SUBAPPLICATION AR2_TAP_TO_AR (* Zapft einen zusaetzlichen Nur-Lese-Pfad (AR_OUT, plain AR) aus einer bestehenden AR2-Verbindung ab, ohne deren urspruengliche Persistenz-/Restore-Kette zu unterbrechen. Socket AR2_IN haengt an die Quelle (einen bestehenden AR2-Plug, z.B. AR_CALIBRATE_2P_REF.X_LOW), Plug AR2_OUT fuehrt die AR2-Verbindung unveraendert zum urspruenglichen Ziel weiter (einen bestehenden AR2-Socket, z.B. INI_AR2.VAL). Kombination aus AR2_TO_AR + AR_SPLIT_2 + AR_TO_AR2 (3 bereits vorhandene Standardbausteine) - kein eigener AR2-Split-Baustein existiert im Projekt, AR2 ist wie jeder Adapter strikt 1:1. *)
  (* Standard: 61499-2; Description: Copyright (c) 2026 Meisterschulen am Ostbahnhof This program and the accompanying materials are made available under the terms of the Eclipse Public License 2.0 which is available at https://www.eclipse.org/legal/epl-2.0/ SPDX-License-Identifier: EPL-2.0 *)
  (* Version 1.0, 2026-09-20, Franz Höpfinger, Meisterschulen am Ostbahnhof, initial implementation - fuer die Rohwert-Anzeige (Zero/Span bzw. Min/Mid/Max Raw) in logiBUS_AI_Calibrate_IDA_OPC/_3P_IDA_OPC (Button_AI_Calibrate_OPC_UA/_3P_OPC_UA): AR_CALIBRATE_2P_REF/_3P_REF speichern X_LOW/X_HIGH bzw. X_MIN/X_MID/X_MAX bereits als AR2-Plugs, bisher aber nur an die INI-Persistierung angeschlossen, nirgends zur Anzeige. *)
  PACKAGE MyLib::sys;
  (* Documentation:
  AR2_TAP_TO_AR
   🇩🇪 Deutsch
   Haengt zwischen eine bestehende AR2-Plug/Socket-Verbindung, ohne deren Verhalten zu aendern, und liefert zusaetzlich einen Nur-Lese-Spiegel (AR_OUT, plain AR) des aktuellen Werts.
   Warum nicht einfach splitten?
   Adapter sind strikt 1:1 - ein Plug wie AR_CALIBRATE_2P_REF.X_LOW kann nur an EINEN Socket angeschlossen werden. Fuer unidirektionale Adapter (AR/AX) gibt es dafuer AR_SPLIT_2/AX_SPLIT_2 usw. - fuer bidirektionale AR2 existiert kein aequivalenter Split-Baustein im Projekt, da AR2 normalerweise genau 1 Erzeuger und genau 1 Verbraucher hat.
   Wie es funktioniert
   AR2_TO_AR (Socket AR2_BIDIR, haengt an die Quelle) spiegelt die von der Quelle geschriebene Seite nach AR_OUT - dieser Wert wird per AR_SPLIT_2 aufgeteilt: einmal nach aussen (AR_OUT dieses Bausteins, fuer die Anzeige), einmal in AR_TO_AR2 (Socket AR_IN), das daraus wieder eine vollwertige AR2-Verbindung macht (Plug AR2_BIDIR, geht weiter zum urspruenglichen Ziel, z.B. INI_AR2). Der Rueckweg (persistierter/restaurierter Wert von INI_AR2) laeuft symmetrisch zurueck: AR_TO_AR2.AR_OUT speist AR2_TO_AR.AR_IN, wodurch die Quelle (AR_CALIBRATE_2P_REF.X_LOW) ihren Restore-Wert weiterhin ganz normal ueber EI1/DI1 bekommt - nichts an der urspruenglichen Kette aendert sich, es kommt nur ein Abzweig hinzu.
   🇬🇧 English
   Sits between an existing AR2 Plug/Socket connection without changing its behaviour, and additionally provides a read-only plain-AR mirror (AR_OUT) of the current value.
   Why not just split it?
   Adapters are strictly 1:1 - a Plug like AR_CALIBRATE_2P_REF.X_LOW can only connect to ONE Socket. For unidirectional adapters (AR/AX) there is AR_SPLIT_2/AX_SPLIT_2 etc. for this - no equivalent split block exists for bidirectional AR2 in this project, since AR2 normally has exactly one producer and one consumer.
   How it works
   AR2_TO_AR (Socket AR2_BIDIR, attaches to the source) mirrors the side written by the source out through AR_OUT - this value is split via AR_SPLIT_2: once outward (this block's own AR_OUT, for display), once into AR_TO_AR2 (Socket AR_IN), which turns it back into a full AR2 connection (Plug AR2_BIDIR, continues to the original target, e.g. INI_AR2). The return path (persisted/restored value from INI_AR2) runs symmetrically back: AR_TO_AR2.AR_OUT feeds AR2_TO_AR.AR_IN, so the source (AR_CALIBRATE_2P_REF.X_LOW) still gets its restored value normally via EI1/DI1 - nothing about the original chain changes, only a tap is added.
  *)
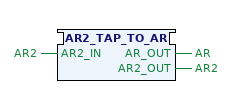
  SOCKETS
    AR2_IN : adapter::types::bidirectional::AR2; (* Haengt an die AR2-Quelle (Plug), z.B. AR_CALIBRATE_2P_REF.X_LOW *)
  END_SOCKETS
  PLUGS
    AR_OUT : adapter::types::unidirectional::AR; (* Nur-Lese-Spiegel des aktuellen Werts (neu geschriebener Wert sofort, persistierter/restaurierter Wert nach Boot) - fuer VT-Anzeige/OPC-UA-Publish *)
    AR2_OUT : adapter::types::bidirectional::AR2; (* Fuehrt die AR2-Verbindung unveraendert weiter zum urspruenglichen Ziel (Socket), z.B. INI_AR2.VAL *)
  END_PLUGS
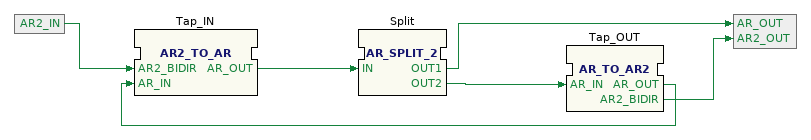
  FBS
    Tap_IN : adapter::conversion::bidirectional::AR2_TO_AR;
    Split : adapter::events::unidirectional::AR_SPLIT_2;
    Tap_OUT : adapter::conversion::bidirectional::AR_TO_AR2;
  END_FBS
  ADAPTER_CONNECTIONS
    AR2_IN TO Tap_IN.AR2_BIDIR;
    Tap_OUT.AR_OUT TO Tap_IN.AR_IN;
    Tap_IN.AR_OUT TO Split.IN;
    Split.OUT1 TO AR_OUT;
    Split.OUT2 TO Tap_OUT.AR_IN;
    Tap_OUT.AR2_BIDIR TO AR2_OUT;
  END_CONNECTIONS
END_SUBAPPLICATION
